FUNCTION Convert_DWORD_TO_SINT : Hresult
VAR_INPUT
	in : DWORD;
	out : REFERENCE TO SINT;
END_VAR
VAR
	converted : SINT;
END_VAR
VAR CONSTANT
	INCOMPATIBLE : HRESULT := 16#9811070E;
END_VAR

converted := DWORD_TO_SINT(in);

IF (SINT_TO_DWORD(converted) <> in) THEN
	Convert_DWORD_TO_SINT := INCOMPATIBLE;
	RETURN;
END_IF

out := converted;

END_FUNCTION

(* stored: Version 1.1.0.1, ProductVersion 3.1.4024.12
   POU Convert_DWORD_TO_SINT: Id {acaef23d-f7d5-4a9b-8ac6-87e95df587da}, SpecialFunc None *)
